Staubli VAL3: checkTrackArea.pgx

public program checkTrackArea(tool x_tActivTool, num& x_nWrkZone[])
  local trsf l_trToolPos
begin
  // This program checks if the robot is inside the Tracking window
  //
  // Input Param
  // x_tActivTool  : TCP to ckeck position
  //
  // Output Param
  // x_nWrkZone : real value
  //          0 --> Beside conveyor
  //          1 --> Upstream of the upstream end of the tracking window.
  //          2 --> Within the tracking window
  //          3 --> Downstream of the downstream end of the tracking window.
  //
  // Created 07-03-08                                   C.CURRIVAND
  //----------------------------------------------------------------
  //
  l_trToolPos=position(here(x_tActivTool,fConveyor),fConveyor)
  //
  x_nWrkZone=0
  //Check Z coordinate
  if (abs(l_trToolPos.z)<nTrackWinHeight)
    // ----- Check robot position against upstream end
    // check Y coordinate
    if (l_trToolPos.y>=trBoundaryUp[0].y) and (l_trToolPos.y<=trBoundaryUp[1].y)
      // Y is OK, check X coordinate
      if nA1==0
        x_nWrkZone=sel(l_trToolPos.x>trBoundaryUp[0].x,2,1)
      elseIf nA1>0
        x_nWrkZone=sel(l_trToolPos.y<nA1*l_trToolPos.x+nB1,2,1)
      elseIf nA1<0
        x_nWrkZone=sel(l_trToolPos.y>nA1*l_trToolPos.x+nB1,2,1)
      endIf
    endIf
    // Robot is downstream of upstream limit
    //---- Check robot position against downstream end
    if x_nWrkZone==2
      // check Y coordinate
      if (l_trToolPos.y>=trBoundaryDwn[0].y) and (l_trToolPos.y<=trBoundaryDwn[1].y)
        // Y is OK, check X coordinate
        if nA2==0
          x_nWrkZone=sel(l_trToolPos.x<=trBoundaryDwn[0].x,2,3)
        elseIf nA2>0
          x_nWrkZone=sel(l_trToolPos.y>nA2*l_trToolPos.x+nB2,2,3)
        elseIf nA2<0
          x_nWrkZone=sel(l_trToolPos.y<nA2*l_trToolPos.x+nB2,2,3)
        endIf
      endIf
    endIf
  endIf
end
